FUNCTION_BLOCK CL_WorkbenchSensor
VAR_INPUT
END_VAR
VAR_OUTPUT
END_VAR
VAR
  bInit : BOOL := FALSE;
  _bSensorRaw_P:  POINTER TO BOOL;
  timeFilter: TON;
  risEdgeDetector:  R_TRIG;
END_VAR

METHOD Init : BOOL
VAR_INPUT
  bSensor_P:  POINTER TO BOOL;
END_VAR
IF (bInit = FALSE) AND (bSensor_P <> 0) THEN
  timeFilter.PT := T#100MS;
  _bSensorRaw_P := bSensor_P;
  bInit := TRUE;
END_IF
END_METHOD

METHOD PUBLIC isModule : BOOL
VAR_INPUT
END_VAR

VAR
  filteredSensor: BOOL;
END_VAR
timeFilter(IN:=_bSensorRaw_P^,PT:=T#100MS,Q=>filteredSensor); // True if signal maintained to 1 long enough
risEdgeDetector(CLK:=filteredSensor,Q=>isModule); // True at the exact rise detection
END_METHOD

END_FUNCTION_BLOCK

(* stored: Version 1.1.0.1, ProductVersion 3.1.4024.12
   POU CL_WorkbenchSensor: Id {7186c0f7-0441-4f85-ac29-deaaa6783b1d}, SpecialFunc None
   Method Init: Id {27f678ec-63b0-4f0e-9c9d-eb8fb196e2f3}
   Method isModule: Id {7e31d7fd-ccaf-496b-ac31-2c1f82e8cf37} *)
